{attribute 'qualified_only'}
{attribute 'strict'}
{attribute 'to_string'}
TYPE E_PizzaOvenStates :
(
	WaitForPizzaInOven 	:= 0,
	WeJustGotAPizza		:= 1,
	MovePizzaOutOfOven	:= 2
);
END_TYPE

(* stored: Version 1.1.0.1
   DUT E_PizzaOvenStates: Id {47d5b72e-96cb-4abb-83d1-05bfff017557} *)
